TYPE Controller :
STRUCT
	bDpadRight : BOOL;
	bDpadLeft : BOOL;
	bDpadUp : BOOL;
	bDpadDown : BOOL;
	bAbtn : BOOL;
	bBbtn : BOOL;
	bXbtn : BOOL;
	bYbtn : BOOL;
	rightStick : ARRAY[0..2] OF REAL;
	leftStick : ARRAY[0..2] OF REAL;
END_STRUCT
END_TYPE

(* stored: Version 1.1.0.1, ProductVersion 3.1.4024.9
   DUT Controller: Id {1116ce3c-e681-4f9e-b11f-1f70e96e06b2} *)
